TYPE ST_LAB_PackData :
STRUCT
	sPackCode			: T_MaxString;
	nPackStatus			: INT;
	nPackRejectID		: UINT;
END_STRUCT
END_TYPE

(* stored: Version 1.1.0.1
   DUT ST_LAB_PackData: Id {172e89ca-c344-458f-beb2-ab9cb7a0c8e2} *)
